(* PLC project CoDeSys External Library Template, WAGO e!COCKPIT e!COCKPIT, author 3S - Smart Software Solutions GmbH *)
(* stored: creationDateTime 2019-10-29T12:22:40.9690023, version 3.5.5.30, modificationDateTime 2019-10-24T14:40:07.960949, organization 3S - Smart Software Solutions GmbH *)
(* Library project template with all possible element types, docu and a sample project structure *)

FUNCTION fnOdwrocenieBitowTemperaturyUjemnejREAL_TO_WORD : WORD
  VAR_INPUT
    rTemperaturaKelviny : REAL;
  END_VAR

            (*			
Autor:					Artur Wyszomirski, 2019-05-27 
Prawa majątkowe: 		Solwena Sp. z o.o., 
Aktualizacje:			 
					
Opis:					Funkcja odwraca bity temperatury, jeśli tempratura jest mniejsza ujemna w skali Celsjusza. Wartość wejściowa w REAL, wartość wyjściowa w WORD.
*)
IF rTemperaturaKelviny < 273.15 THEN	// Jeśli temperatura jest ujemna, odwróć bity
	fnOdwrocenieBitowTemperaturyUjemnejREAL_TO_WORD := REAL_TO_WORD(65535 - (ABS(rTemperaturaKelviny - 273.15) * 10));	
ELSE
	fnOdwrocenieBitowTemperaturyUjemnejREAL_TO_WORD := REAL_TO_WORD((rTemperaturaKelviny - 273.15) * 10);						
END_IF
          
END_FUNCTION
